PROGRAM Qrob_control

VAR_INPUT
	
	aux_cu :REAL;
	reset : bool;
	external : BOOL;
    mover_horario:	BOOL;
	mover_antihorario: BOOL;
	velocidad: REAL := 10 ;
	velocidad_ext: REAL := 100 ;
	set_posicion_mover :INT := 25;
	EnableAxis1 : BOOL := TRUE;
	detener : BOOL;
	mover_abs :BOOL;
	pos_mover_abs :REAL ;
	
	ajustar_tornillo : BOOL ;
	limite_corriente : REAL := 120;
	torque_relief : BOOL := FALSE;
	tor_on : BOOL;
    tor_val : INT;
		aux_velo : BOOL;
	
END_VAR

VAR
	
	fbPower: MC_Power;
	Axis1Enabled : BOOL;
	actual_position : LREAL;
	actual_velocity : REAL;
	original_vel :DINT;
	actual_current  :  LREAL;
	position_ok :BOOL;
	home :	 BOOL;
	mov_abs_ok : BOOL;
	max_current : BOOL;
	val_max_current : REAL;
	aux_current : REAL;

	
	MC_Home: MC_HOME;
	MC_ReadActualPosition: MC_ReadActualPosition;
	MC_ReadActualVelocity : MC_ReadActualVelocity;
	MC_ReadParameter_0: MC_ReadParameter;
	MC_MoveVelocity_horario: MC_MoveVelocity;
	MC_MoveVelocity_antiorario: MC_MoveVelocity;
	MC_Stop: MC_Stop;
	MC_Stop2: MC_Stop;
	MC_MoveAbsolute: MC_MoveAbsolute;
    MC_TorqueControl : MC_TorqueControl;
	Ton : TON;
	RS : RS;
	limit_current : limit_current;
	
	
	fuzzy : Subsystem;
	fuzzy_vel : LREAL;
	fuzzy_active : BOOL;
	stop_limit : BOOL;
    MC_ExtSetPointGenEnable : MC_ExtSetPointGenEnable;
	MC_Reset : MC_Reset;
	MC_MoveSuperImposed : MC_MoveSuperImposed;
    FB_CTRL_SETPOINT_GENERATOR : FB_CTRL_SETPOINT_GENERATOR;

	num_ran : LREAL;
	pulse : BOOL:= TRUE;
	PT_b : BOOL;
	DRAND : DRAND;
	pulse1 : pulse_;
	nrand_out : LREAL;
   
	state_move_active : BOOL;	
	
	
END_VAR

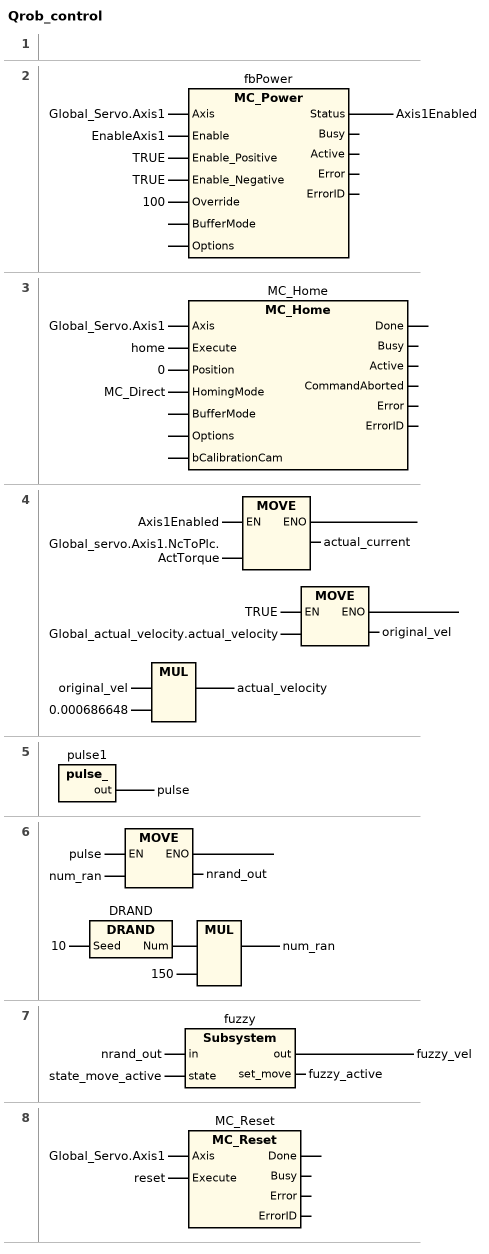
// NETWORK 1

// NETWORK 2
fbPower(
    Axis := Global_Servo.Axis1,
    Enable := EnableAxis1,
    Enable_Positive := TRUE,
    Enable_Negative := TRUE,
    Override := 100); // MC_Power
Axis1Enabled := fbPower.Status;

// NETWORK 3
MC_Home(Axis := Global_Servo.Axis1, Execute := home, Position := 0, HomingMode := MC_Direct);

// NETWORK 4
IF Axis1Enabled THEN actual_current := Global_servo.Axis1.NcToPlc.ActTorque; END_IF
original_vel := Global_actual_velocity.actual_velocity;
actual_velocity := original_vel * 0.000686648;

// NETWORK 5
pulse1(); // pulse_
pulse := pulse1.out;

// NETWORK 6
IF pulse THEN nrand_out := num_ran; END_IF
DRAND(Seed := 10);
num_ran := DRAND.Num * 150;

// NETWORK 7
fuzzy(in := nrand_out, state := state_move_active, set_move => fuzzy_active); // Subsystem
fuzzy_vel := fuzzy.out;

// NETWORK 8
MC_Reset(Axis := Global_Servo.Axis1, Execute := reset);

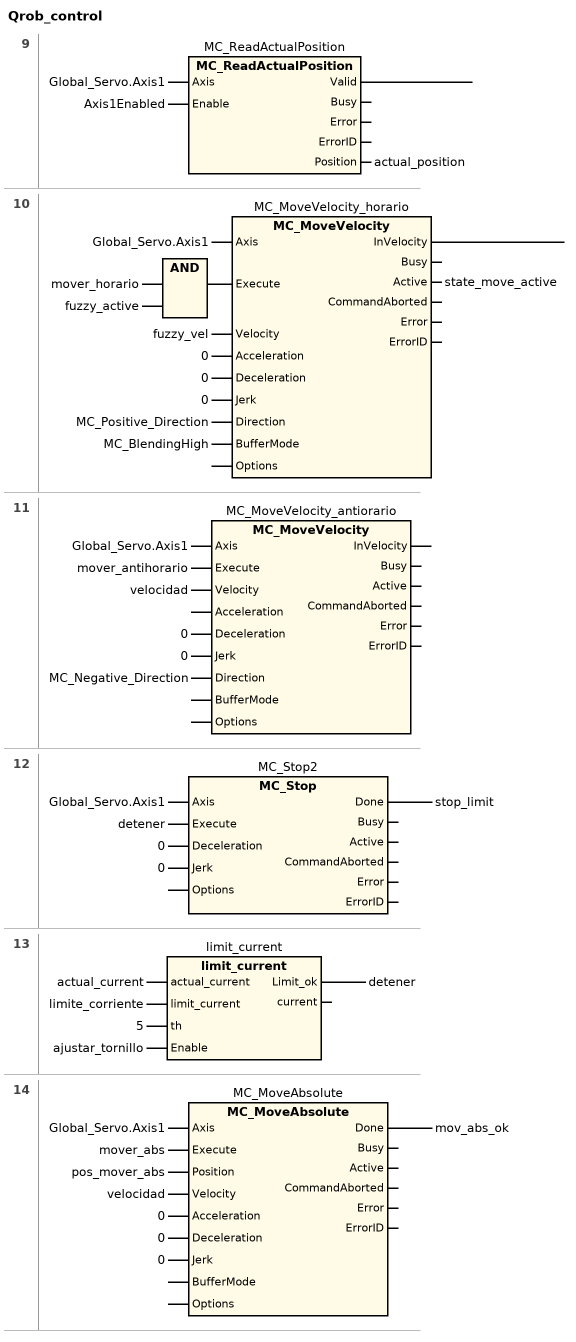
// NETWORK 9
MC_ReadActualPosition(Axis := Global_Servo.Axis1, Enable := Axis1Enabled, Position => actual_position);

// NETWORK 10
MC_MoveVelocity_horario(
    Axis := Global_Servo.Axis1,
    Execute := mover_horario AND fuzzy_active,
    Velocity := fuzzy_vel,
    Acceleration := 0,
    Deceleration := 0,
    Jerk := 0,
    Direction := MC_Positive_Direction,
    BufferMode := MC_BlendingHigh,
    Active => state_move_active); // MC_MoveVelocity

// NETWORK 11
MC_MoveVelocity_antiorario(
    Axis := Global_Servo.Axis1,
    Execute := mover_antihorario,
    Velocity := velocidad,
    Deceleration := 0,
    Jerk := 0,
    Direction := MC_Negative_Direction); // MC_MoveVelocity

// NETWORK 12
MC_Stop2(Axis := Global_Servo.Axis1, Execute := detener, Deceleration := 0, Jerk := 0); // MC_Stop
stop_limit := MC_Stop2.Done;

// NETWORK 13
limit_current(
    actual_current := actual_current,
    limit_current := limite_corriente,
    th := 5,
    Enable := ajustar_tornillo);
detener := limit_current.Limit_ok;

// NETWORK 14
MC_MoveAbsolute(
    Axis := Global_Servo.Axis1,
    Execute := mover_abs,
    Position := pos_mover_abs,
    Velocity := velocidad,
    Acceleration := 0,
    Deceleration := 0,
    Jerk := 0);
mov_abs_ok := MC_MoveAbsolute.Done;

END_PROGRAM

(* stored: Version 1.1.0.1, ProductVersion 3.1.4024.4
   POU Qrob_control: Id {8c37094b-a5bd-4eb6-9947-3cb2108e38b7}, SpecialFunc None *)
